{attribute 'GeneratedUsingTerminal: EK1100-0000-0018'}
{attribute addProperty BoxType "EK1100-0000-0018"}
{attribute addProperty Id "Beckhoff_ER1xxxEK1122Beckhoff_ER1xxxEK1122_4914C526508"}
{attribute addProperty CRC "2789082970"}
{attribute addProperty Size "508"}
TYPE Beckhoff_ER1xxx_A63E075A EXTENDS EK1100_1FC0878B :
STRUCT
	{attribute addProperty Name "Beckhoff_ER1xxxEK1122"}
	{attribute addProperty PreviousPort "Beckhoff ER1xxx : B"}
	Beckhoff_ER1xxxEK1122 : Beckhoff_ER1xxxEK1122_4914C526;
END_STRUCT
END_TYPE

(* stored: Version 1.2.0.0, ProductVersion 3.1.4024.9
   DUT Beckhoff_ER1xxx_A63E075A: Id {0a766467-0213-4fcd-97e8-1a53d711d710} *)
